# EPICS autosave request: ESP300/iocBoot/ioc_esp_bmc/auto_positions.req
file "XFM_motor_positions.req",      P=XF:04BMC-ES:, M=DET:1-Ax:Y:Mtr
